INTERFACE ITF_6AxisRobot EXTENDS ITF_Robot

PROPERTY currentFrame : stFrame
GET
END_GET
SET
END_SET
END_PROPERTY

PROPERTY currentFrameID : UINT
GET
END_GET
END_PROPERTY

PROPERTY currentTool : FB_Tool
GET
END_GET
SET
END_SET
END_PROPERTY

METHOD Home : BOOL
VAR_INPUT
END_VAR
END_METHOD

PROPERTY isInCollision : BOOL
GET
END_GET
END_PROPERTY

PROPERTY isInHomePosition : BOOL
GET
END_GET
END_PROPERTY

PROPERTY jointPosition : stJointPosition6
GET
END_GET
END_PROPERTY

PROPERTY jointVelocity : stJointPosition6
GET
END_GET
END_PROPERTY

METHOD SwitchTool : UINT
VAR_INPUT
	tool: FB_Tool;
END_VAR
END_METHOD

PROPERTY TCPPosition : stPose3D
GET
END_GET
END_PROPERTY

PROPERTY TCPVelocity : stPose3D
GET
END_GET
END_PROPERTY

END_INTERFACE

(* stored: Version 1.1.0.1, ProductVersion 3.1.4026.18
   Itf ITF_6AxisRobot: Id {5597e200-2768-442d-a894-79ed17b4bd75}
   Property currentFrame: Id {1b2bad2f-6e4f-4380-af0a-eb03279d228f}
   Get Get: Id {8c170702-04a0-4274-a991-247107592a5b}
   Set Set: Id {2305773b-70ee-4c13-98f5-0ef584f3b9e2}
   Property currentFrameID: Id {9469c945-f6c9-484b-8b35-ecb495593b6d}
   Get Get: Id {012f4be9-5ca5-4a9b-bf63-a841d9320e0f}
   Property currentTool: Id {a924a41c-da33-494b-a68c-a36e519d8e2b}
   Get Get: Id {f1108b85-0eba-49a3-9a34-bb0dc96e56ae}
   Set Set: Id {3f004d9a-8a4f-4c33-adca-e53e42e82a18}
   Method Home: Id {9008c31c-e8e7-4fc4-ab50-fce636f66aa9}
   Property isInCollision: Id {93a59f2f-27ed-4f85-bd2a-37d1c5c6c38a}
   Get Get: Id {70d3b40f-fa30-44f4-b5a6-e57862b63326}
   Property isInHomePosition: Id {68f1d365-ed87-4b19-84e6-4cf49a3eac85}
   Get Get: Id {08952083-8143-4845-a361-fe2a403fa7ce}
   Property jointPosition: Id {967eac40-c236-4e95-bd58-25ccf022c448}
   Get Get: Id {0e471fba-f0f4-49f8-bf46-53a8148575e4}
   Property jointVelocity: Id {a5ea3d6b-243a-4425-9bdd-13270e6b23d8}
   Get Get: Id {b2cbd5f6-df64-4021-8c9b-d68ee343f3fa}
   Method SwitchTool: Id {4419060a-b81d-49ba-98b5-0e9531683def}
   Property TCPPosition: Id {5e92b5b7-e827-4b57-8516-68a57c3f5a78}
   Get Get: Id {d87b70c6-fddf-466e-a406-eede7e052a5f}
   Property TCPVelocity: Id {29c2cbff-861a-434c-bd80-cca88e4b0432}
   Get Get: Id {d62f14c4-b447-4702-98b3-1685b412e392} *)
